(* Schneider Machine Expert - Basic project Questao3.7_FelipeV1_20241014, file version 2.9.0.0 *)
(* ProjectInformations: Name=Novo projeto *)

HARDWARE
  Cpu 0: TM221M16R/G
  EthernetConfiguration: NetworkName=M221, IpAllocationMode=FixedAddress, IpAddress=0.0.0.0, SubnetMask=0.0.0.0
  SerialLineConfiguration: Baud=Baud19200, Parity=ParityEven, DataBits=DataBits8, StopBits=StopBits1, PhysicalMedium=PhysicalMediumRs485, TransmissionMode=TransmissionModeModbusRtu, SlaveId=1, Addressing=SlaveAddressing
  MastTask: UsePeriodScanMode=false, PeriodScan=100
  FastTask: Period=255
  CpuBehavior: StartingMode=StartAsPreviousState, AutoSaveRamOnEeprom=true, WatchdogPeriod=250

SYMBOLS  (address, symbol, comment, settings)
  %M0       LED_1
  %M1       TIMER_1
  %M10      ACIO_LED_A
  %TM0      TEMP_1  [Preset=2, Base=OneSecond]
  %I0.0     CONT_LED_A
  %I0.1     CONT_LIGA_TIME_1
  %Q0.0     SAIDA__LED_1

POU Entradas
  (* SectionNumber=1 *)

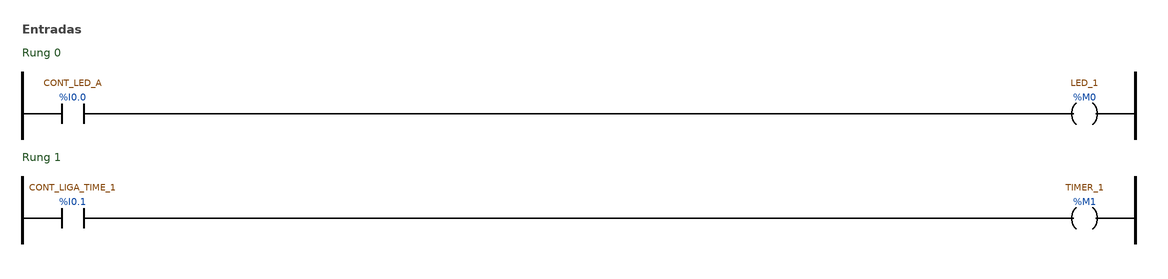

// Rung 0
  LD %I0.0                (* CONT_LED_A *)
  ST %M0                  (* LED_1 *)
  // as ST:
  //   LED_1 := CONT_LED_A;

// Rung 1
  LD %I0.1                (* CONT_LIGA_TIME_1 *)
  ST %M1                  (* TIMER_1 *)
  // as ST:
  //   TIMER_1 := CONT_LIGA_TIME_1;

POU Lógica
  (* SectionNumber=2 *)

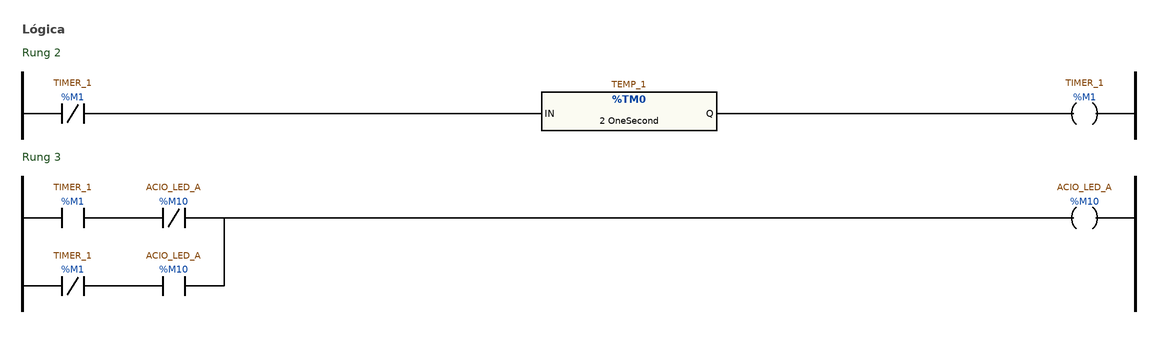

// Rung 2
  BLK %TM0                (* TEMP_1 *)
  LDN %M1                 (* TIMER_1 *)
  IN
  OUT_BLK
  LD Q
  ST %M1                  (* TIMER_1 *)
  END_BLK
  // as ST:
  //   TEMP_1(IN := NOT TIMER_1);
  //   TIMER_1 := TEMP_1.Q;

// Rung 3
  LD %M1                  (* TIMER_1 *)
  ANDN %M10               (* ACIO_LED_A *)
  OR(N %M1                (* TIMER_1 *)
  AND %M10                (* ACIO_LED_A *)
  )
  ST %M10                 (* ACIO_LED_A *)
  // as ST:
  //   ACIO_LED_A := TIMER_1 AND NOT ACIO_LED_A OR NOT TIMER_1 AND ACIO_LED_A;

POU Saídas
  (* SectionNumber=3 *)

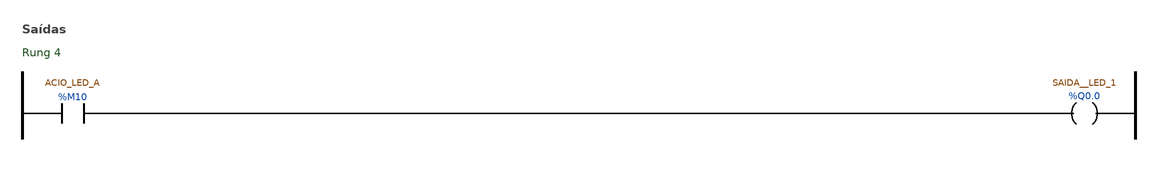

// Rung 4
  LD %M10                 (* ACIO_LED_A *)
  ST %Q0.0                (* SAIDA__LED_1 *)
  // as ST:
  //   SAIDA__LED_1 := ACIO_LED_A;
